{attribute 'linkalways'} 
{attribute 'no_explicit_call' := 'This FB is a CLASS and must be accessed using methods or properties'}
{attribute 'enable_dynamic_creation'}
FUNCTION_BLOCK Node_F_VN_DrawCircle EXTENDS VisionNode
VAR
    nCenterX : _UDINT(0);
    nCenterY : _UDINT(0);
    nRadius : _UDINT(0);
    ipDestImage : _ITcVnImage;
    aColor : _TcVnVector4_LREAL;
    nThickness : _DINT(1);
    hrPrev : _HRESULT(S_OK);
	hresult : _HRESULT(S_OK);
END_VAR

METHOD PUBLIC  Clone : I_Node
VAR
	pNode : POINTER TO Node_F_VN_DrawCircle;
END_VAR
pNode := __NEW(Node_F_VN_DrawCircle);
Clone := pNode^;
END_METHOD

METHOD FB_init : BOOL
VAR_INPUT
	bInitRetains : BOOL; // if TRUE, the retain variables are initialized (warm start / cold start)
	bInCopyCode : BOOL;  // if TRUE, the instance afterwards gets moved into the copy code (online change)
END_VAR
AddParameter('nCenterX', nCenterX);
AddParameter('nCenterY', nCenterY);
AddParameter('nRadius', nRadius);
AddInput('ipDestImage', ipDestImage);
AddInput('aColor', aColor);
AddParameter('nThickness', nThickness);
AddInput('hrPrev', hrPrev);
AddOutput('ipDestImage', ipDestImage);
AddOutput('hresult',hresult);
END_METHOD

METHOD PROTECTED OnExecute
hresult.Value := F_VN_DrawCircle(
    nCenterX := nCenterX.Value,
    nCenterY := nCenterY.Value,
    nRadius := nRadius.Value,
	ipDestImage := ipDestImage.Value,
    aColor := aColor.Value,
    nThickness := nThickness.Value,
	hrPrev:= hrPrev.Value);
END_METHOD

METHOD PUBLIC PreExecutionCheck
VAR_INPUT
	Check : I_PreExecutionChecks;
END_VAR
Check.IsTrue(ipDestImage.IsValid, 'ipDestImage must contain an image');
Check.IsTrue(nThickness.Value <> 0, 'nThickness must be non-zero');
END_METHOD

END_FUNCTION_BLOCK

(* stored: Version 1.1.0.1, ProductVersion 3.1.4024.15
   POU Node_F_VN_DrawCircle: Id {d9a62f1e-e3bb-0392-326e-34ccd3c7a486}, SpecialFunc None
   Folder Constructor: Id {cbc1569c-a94e-0fd5-07c7-43e1e64565cc}
   Method Clone: Id {570236a5-5b7b-030e-00da-c33498d23061}
   Method FB_init: Id {6f8c1798-8dfc-0c6c-1f29-1d44954dba0b}
   Method OnExecute: Id {15a910b2-c59d-00da-041a-c5dc11c496c9}
   Method PreExecutionCheck: Id {3aec8126-88f2-076b-079e-76d5ac035d88} *)
